FUNCTION_BLOCK LavadoCircuitoLiquidos
VAR_INPUT
	bModoEco:BOOL;
	rCaudalLlenado:REAL;
	rCaudalVaciado:REAL;
	bBomba_enMarcha:BOOL;
	rVelocBombaVaciado:REAL;
	rVelocBombaLavado:REAL;
	tSetTmrVaciado:TIME;
	tSetTmrLlenado:TIME;
	iCantCiclosECO:INT;
	iCantCiclosLavado:INT;
	wEstadoV_AguaResidual:WORD;//bit1=cerrada  bit0=abierta
	wEstadoV_Agua:WORD;//bit1=cerrada  bit0=abierta
	wEstadoCal_V1:WORD;//bit1=a inyeccion  bit0=a probeta
	wEstadoV1:WORD;//bit1=cerrada  bit0=abierta
	wEstadoV2:WORD;//bit1=a proceso  bit0=a limpieza
	wEstadoV3:WORD;//bit1=a agua  bit0=a agua residual
	
END_VAR
VAR_OUTPUT
	rPorcCiclosECO:REAL;
	rPorcCiclosLavado:REAL;
	rPorcAvance:REAL;
	bCa_V1_aProbeta:BOOL;
	bV1_Abrir:BOOL;
	bV2_aLimpieza:BOOL;
	bV3_aResidual:BOOL;
	bV_Residual:BOOL;
	bV_Agua:BOOL;
	rSetVelocBomba:REAL;
	bMarchaBomba:BOOL;
	bReverseBomba:BOOL;

	
END_VAR
VAR_IN_OUT
	bInicioLavado:BOOL;	
	bCancelar:BOOL;
END_VAR
VAR
	TON_Vaciado: TON;
	FinVaciado:BOOL;
	VaciarCircuito:BOOL;
	FinLlenado:BOOL;
	LlenarCircuito:BOOL;
	LavadoLlenar:BOOL;
	LavadoVaciar:BOOL;
	TON_Llenado: TON;
	BombaForward:BOOL;
	BombaReverse:BOOL;
	CtrCiclosModoECO:INT;
	CtrCiclosLavado:INT;
	SetTotalCiclos:REAL;
	TotalCiclosActual:INT;
	rAux:REAL;
	TON_llenadoProbeta: TON;
	TON_vaciadoProbeta: TON;
END_VAR
VAR // added by the converter: edge detectors and wires of the graphical bodies
    _rt1, _rt2 : R_TRIG;
    _w1, _w2, _w3, _w4, _w5, _w6, _w7, _w8 : BOOL;
END_VAR

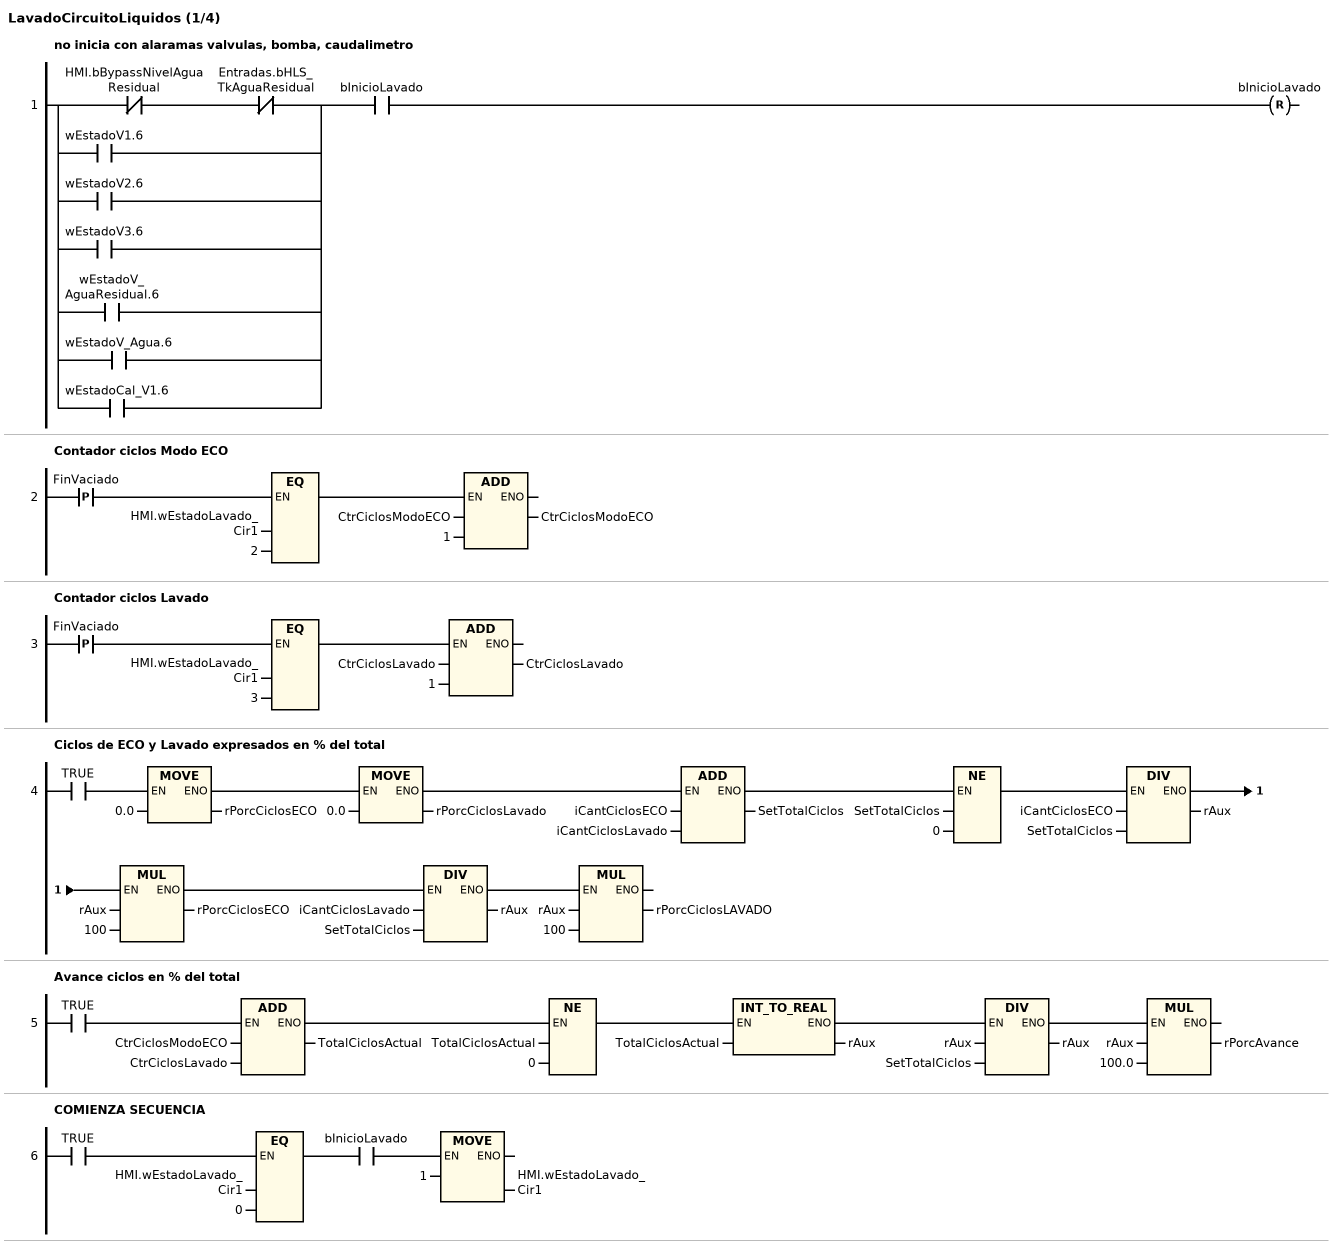
// NETWORK 1: no inicia con alaramas valvulas, bomba, caudalimetro
bInicioLavado R= (NOT HMI.bBypassNivelAguaResidual AND NOT Entradas.bHLS_TkAguaResidual OR wEstadoV1.6 OR wEstadoV2.6 OR wEstadoV3.6 OR wEstadoV_AguaResidual.6 OR wEstadoV_Agua.6 OR wEstadoCal_V1.6) AND bInicioLavado;

// NETWORK 2: Contador ciclos Modo ECO
_rt1(CLK := FinVaciado);
IF _rt1.Q AND HMI.wEstadoLavado_Cir1 = 2 THEN CtrCiclosModoECO := CtrCiclosModoECO + 1; END_IF

// NETWORK 3: Contador ciclos Lavado
_rt2(CLK := FinVaciado);
IF _rt2.Q AND HMI.wEstadoLavado_Cir1 = 3 THEN CtrCiclosLavado := CtrCiclosLavado + 1; END_IF

// NETWORK 4: Ciclos de ECO y Lavado expresados en % del total
rPorcCiclosECO := 0.0;
rPorcCiclosLavado := 0.0;
SetTotalCiclos := iCantCiclosECO + iCantCiclosLavado;
_w1 := SetTotalCiclos <> 0;
IF _w1 THEN rAux := iCantCiclosECO / SetTotalCiclos; END_IF
IF _w1 THEN rPorcCiclosECO := rAux * 100; END_IF
IF _w1 THEN rAux := iCantCiclosLavado / SetTotalCiclos; END_IF
IF _w1 THEN rPorcCiclosLAVADO := rAux * 100; END_IF

// NETWORK 5: Avance ciclos en % del total
TotalCiclosActual := CtrCiclosModoECO + CtrCiclosLavado;
_w2 := TotalCiclosActual <> 0;
IF _w2 THEN rAux := INT_TO_REAL(TotalCiclosActual); END_IF
IF _w2 THEN rAux := rAux / SetTotalCiclos; END_IF
IF _w2 THEN rPorcAvance := rAux * 100.0; END_IF

// NETWORK 6: COMIENZA SECUENCIA
IF HMI.wEstadoLavado_Cir1 = 0 AND bInicioLavado THEN HMI.wEstadoLavado_Cir1 := 1; END_IF

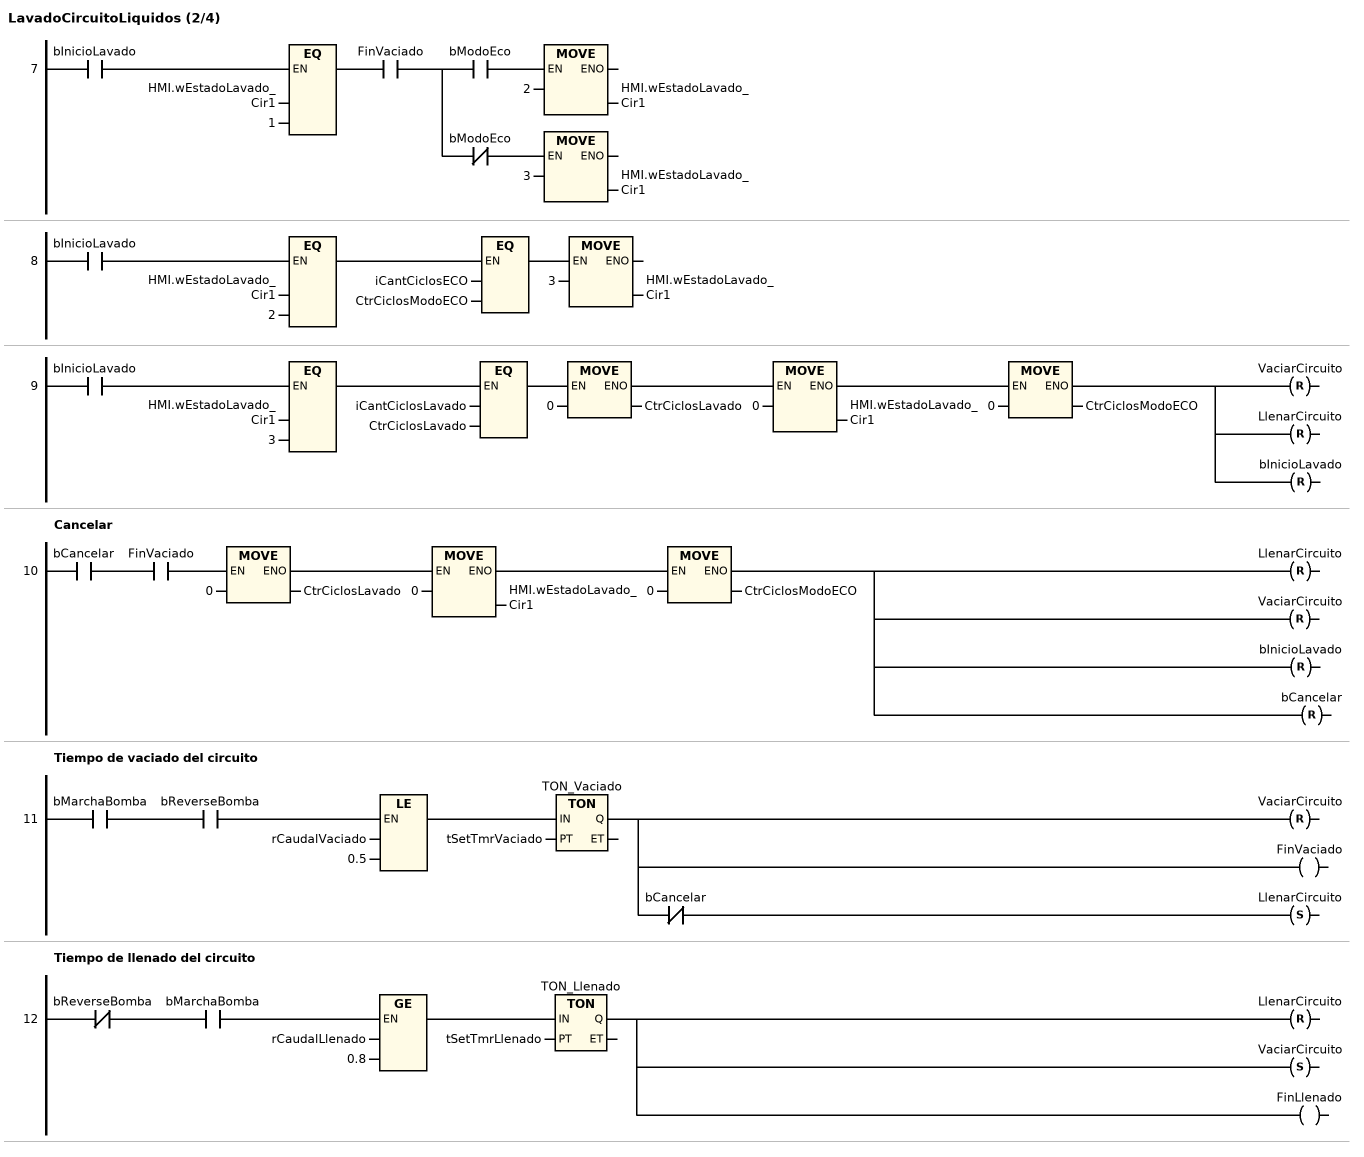
// NETWORK 7
_w3 := (bInicioLavado AND HMI.wEstadoLavado_Cir1 = 1) AND FinVaciado;
IF _w3 AND bModoEco THEN HMI.wEstadoLavado_Cir1 := 2; END_IF
IF _w3 AND NOT bModoEco THEN HMI.wEstadoLavado_Cir1 := 3; END_IF

// NETWORK 8
IF bInicioLavado AND HMI.wEstadoLavado_Cir1 = 2 AND iCantCiclosECO = CtrCiclosModoECO THEN
    HMI.wEstadoLavado_Cir1 := 3;
END_IF

// NETWORK 9
_w4 := bInicioLavado AND HMI.wEstadoLavado_Cir1 = 3 AND iCantCiclosLavado = CtrCiclosLavado;
IF _w4 THEN CtrCiclosLavado := 0; END_IF
IF _w4 THEN HMI.wEstadoLavado_Cir1 := 0; END_IF
IF _w4 THEN CtrCiclosModoECO := 0; END_IF
VaciarCircuito R= _w4;
LlenarCircuito R= _w4;
bInicioLavado R= _w4;

// NETWORK 10: Cancelar
_w5 := bCancelar AND FinVaciado;
IF _w5 THEN CtrCiclosLavado := 0; END_IF
IF _w5 THEN HMI.wEstadoLavado_Cir1 := 0; END_IF
IF _w5 THEN CtrCiclosModoECO := 0; END_IF
LlenarCircuito R= _w5;
VaciarCircuito R= _w5;
bInicioLavado R= _w5;
bCancelar R= _w5;

// NETWORK 11: Tiempo de vaciado del circuito
TON_Vaciado(IN := bMarchaBomba AND bReverseBomba AND rCaudalVaciado <= 0.5, PT := tSetTmrVaciado); // TON
VaciarCircuito R= TON_Vaciado.Q;
FinVaciado := TON_Vaciado.Q;
LlenarCircuito S= TON_Vaciado.Q AND NOT bCancelar;

// NETWORK 12: Tiempo de llenado del circuito
TON_Llenado(IN := NOT bReverseBomba AND bMarchaBomba AND rCaudalLlenado >= 0.8, PT := tSetTmrLlenado); // TON
LlenarCircuito R= TON_Llenado.Q;
VaciarCircuito S= TON_Llenado.Q;
FinLlenado := TON_Llenado.Q;

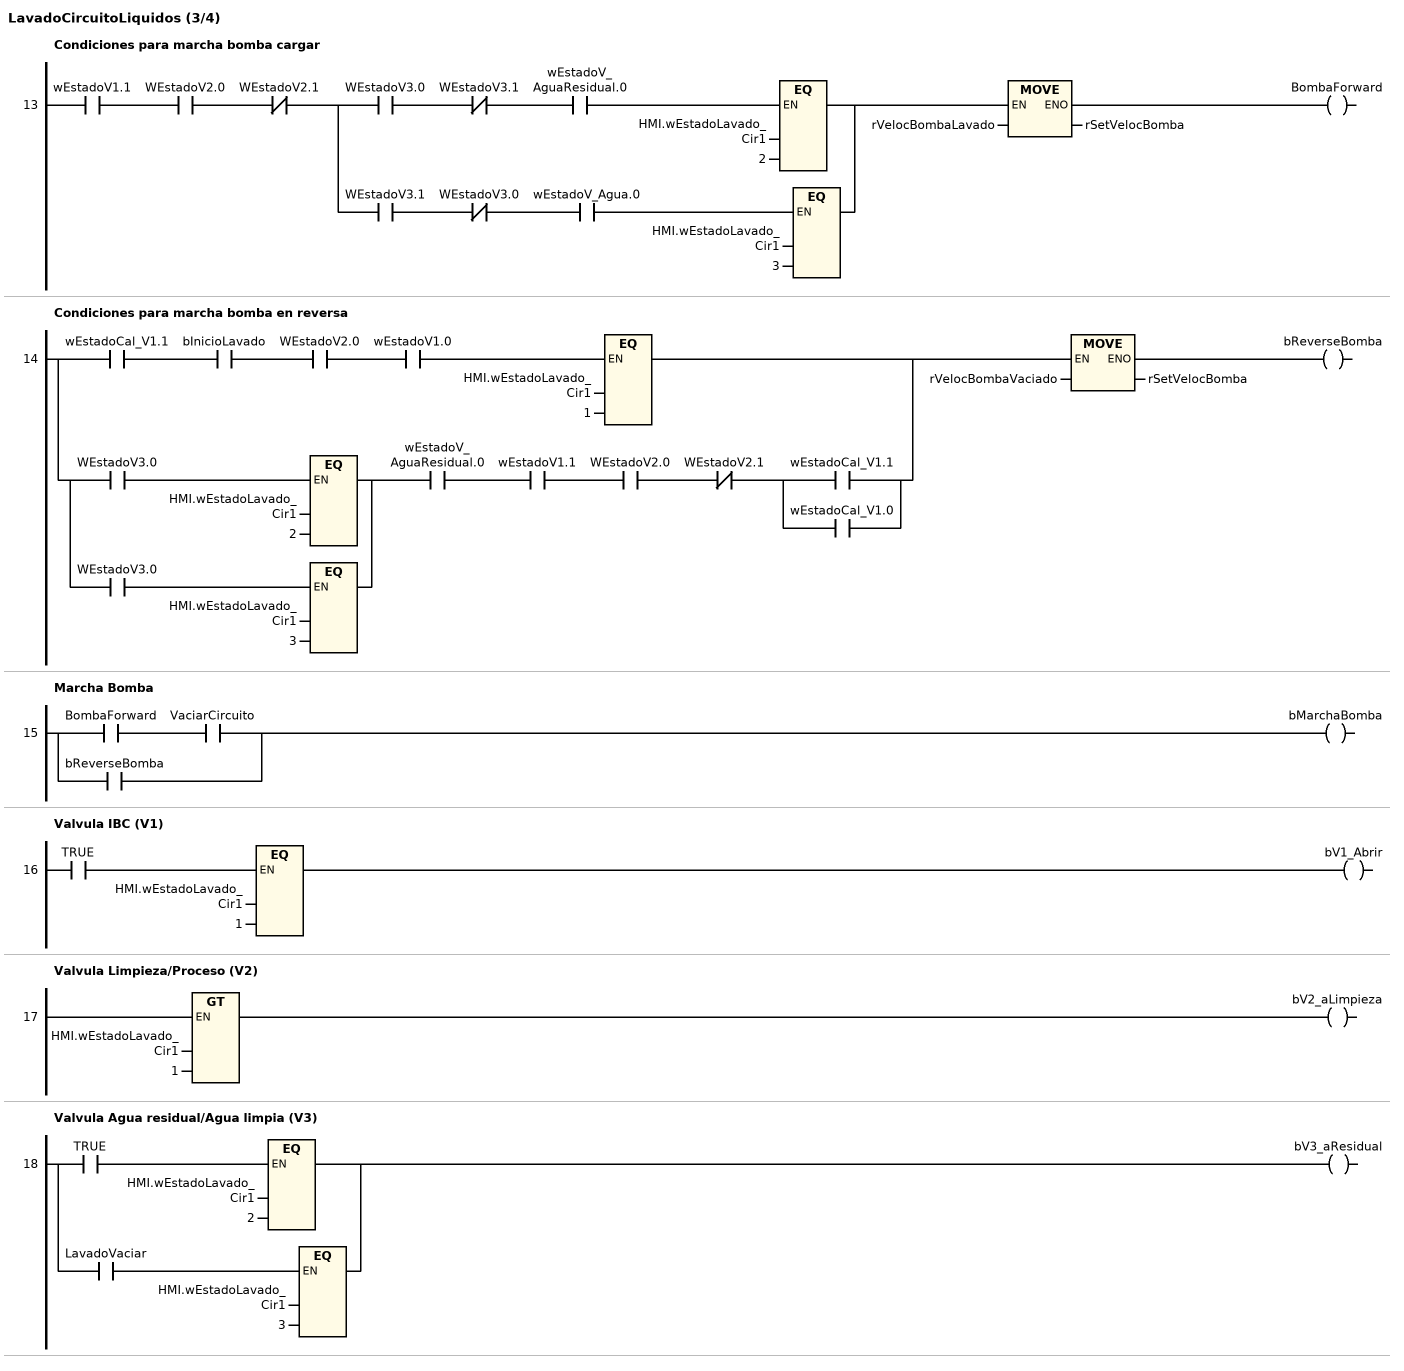
// NETWORK 13: Condiciones para marcha bomba cargar
_w6 := wEstadoV1.1 AND WEstadoV2.0 AND NOT WEstadoV2.1;
_w7 := (_w6 AND WEstadoV3.0) AND NOT WEstadoV3.1 AND wEstadoV_AguaResidual.0 AND HMI.wEstadoLavado_Cir1 = 2 OR (_w6 AND WEstadoV3.1) AND NOT WEstadoV3.0 AND wEstadoV_Agua.0 AND HMI.wEstadoLavado_Cir1 = 3;
IF _w7 THEN rSetVelocBomba := rVelocBombaLavado; END_IF
BombaForward := _w7;

// NETWORK 14: Condiciones para marcha bomba en reversa
_w8 := wEstadoCal_V1.1 AND bInicioLavado AND WEstadoV2.0 AND wEstadoV1.0 AND HMI.wEstadoLavado_Cir1 = 1 OR (WEstadoV3.0 AND HMI.wEstadoLavado_Cir1 = 2 OR WEstadoV3.0 AND HMI.wEstadoLavado_Cir1 = 3) AND wEstadoV_AguaResidual.0 AND wEstadoV1.1 AND WEstadoV2.0 AND NOT WEstadoV2.1 AND (wEstadoCal_V1.1 OR wEstadoCal_V1.0);
IF _w8 THEN rSetVelocBomba := rVelocBombaVaciado; END_IF
bReverseBomba := _w8;

// NETWORK 15: Marcha Bomba
bMarchaBomba := BombaForward AND VaciarCircuito OR bReverseBomba;

// NETWORK 16: Valvula IBC (V1)
bV1_Abrir := HMI.wEstadoLavado_Cir1 = 1;

// NETWORK 17: Valvula Limpieza/Proceso (V2)
bV2_aLimpieza := HMI.wEstadoLavado_Cir1 > 1;

// NETWORK 18: Valvula Agua residual/Agua limpia (V3)
bV3_aResidual := HMI.wEstadoLavado_Cir1 = 2 OR LavadoVaciar AND HMI.wEstadoLavado_Cir1 = 3;

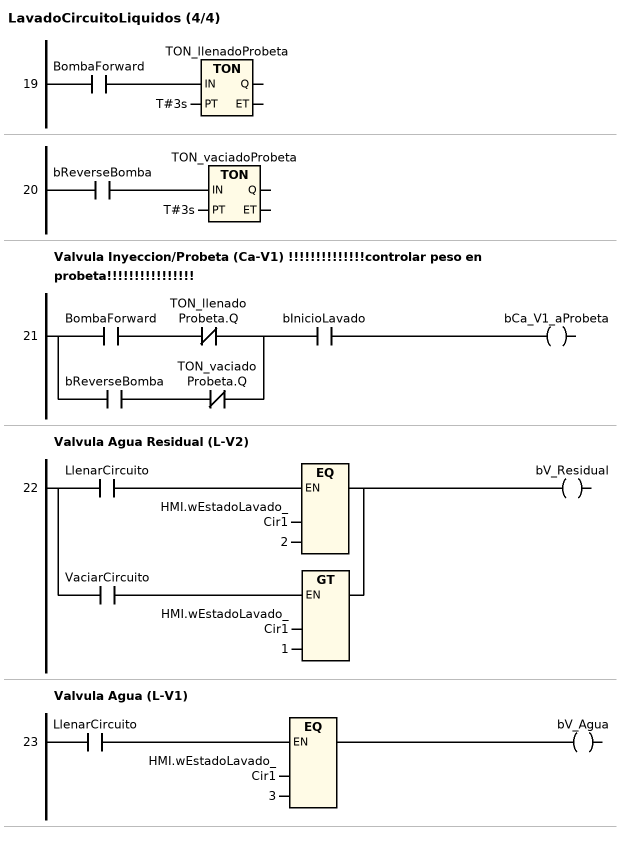
// NETWORK 19
TON_llenadoProbeta(IN := BombaForward, PT := T#3s); // TON

// NETWORK 20
TON_vaciadoProbeta(IN := bReverseBomba, PT := T#3s); // TON

// NETWORK 21: Valvula Inyeccion/Probeta (Ca-V1) !!!!!!!!!!!!!!controlar peso en probeta!!!!!!!!!!!!!!!!
bCa_V1_aProbeta := (BombaForward AND NOT TON_llenadoProbeta.Q OR bReverseBomba AND NOT TON_vaciadoProbeta.Q) AND bInicioLavado;

// NETWORK 22: Valvula Agua Residual (L-V2)
bV_Residual := LlenarCircuito AND HMI.wEstadoLavado_Cir1 = 2 OR VaciarCircuito AND HMI.wEstadoLavado_Cir1 > 1;

// NETWORK 23: Valvula Agua (L-V1)
bV_Agua := LlenarCircuito AND HMI.wEstadoLavado_Cir1 = 3;

END_FUNCTION_BLOCK

(* stored: Version 1.1.0.1, ProductVersion 3.1.4024.12
   POU LavadoCircuitoLiquidos: Id {c7867d05-ffdd-4ec4-81fb-14ae0409b6cc}, SpecialFunc None *)
